(* CoDeSys 2.3.9.62 project: Cap11_7_Res.pro *)
(* Libraries: Standard.lib 4.10.05 12:14:46, IecSfc.lib*2.6.14 10:37:46 *)

(* Global variable list: Global_Variables *)
VAR_GLOBAL

 (* Entradas *)
	M: BOOL;

      (*Salidas*)
	Rojo: BOOL;    	(* Luz roja*)
	Amarillo:BOOL;	(* Luz amarilla *)
	Verde:BOOL;		(* Luz verde *)

END_VAR

(* POU PLC_PRG, SFC *)
PROGRAM PLC_PRG
VAR

       (* declaración  de temporizadores *)
	TEM_ROJO: TON;
	TEM_AMA: TON;
	TEM_VERDE: TON;

    (* declaración  de contadores *)
	CONTA: CTU;

       (* Variables auxiliares *)
	TVERDE: BOOL;     	(* Fin de temporizazión luz verde *)
	TAMA: BOOL;			(* Fin de temporizazión luz amarillo *)
	TROJO: BOOL;		(* Fin de temporizazión luz roja *)

	valor: INT:=3;			(* Número de ciclos a realizar antes de apagarse *)
END_VAR
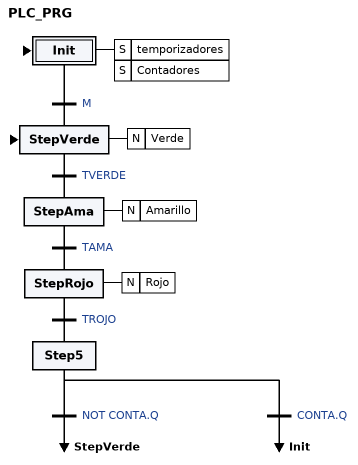
INITIAL_STEP Init:
	temporizadores(S);
	Contadores(S);
END_STEP
TRANSITION FROM Init TO StepVerde := M;
END_TRANSITION
STEP StepVerde:
	Verde(N);
END_STEP
TRANSITION FROM StepVerde TO StepAma := TVERDE;
END_TRANSITION
STEP StepAma:
	Amarillo(N);
END_STEP
TRANSITION FROM StepAma TO StepRojo := TAMA;
END_TRANSITION
STEP StepRojo:
	Rojo(N);
END_STEP
TRANSITION FROM StepRojo TO Step5 := TROJO;
END_TRANSITION
STEP Step5:
END_STEP
TRANSITION FROM Step5 TO StepVerde := NOT CONTA.Q;
END_TRANSITION
TRANSITION FROM Step5 TO Init := CONTA.Q;
END_TRANSITION
END_PROGRAM
ACTION Contadores:
	CAL		CONTA(CU:=StepVerde.x, RESET:=Init.x,PV:=valor)
END_ACTION
ACTION temporizadores:
	CAL		TEM_ROJO(IN:=StepRojo.x, PT:=T#5s, Q=>TROJO)

	CAL		TEM_AMA(IN:=StepAma.x, PT:=T#2s,Q=>TAMA)


	LD		StepVerde.x
	ST		TEM_VERDE.IN
	LD		T#2s
	ST		TEM_VERDE.PT
	CAL		TEM_VERDE
	LD		TEM_VERDE.Q
	ST		TVERDE
END_ACTION

(* Visualisation SemaforoSimple
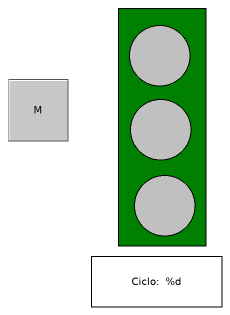
ellipse at (156,41)-(217,102): alarm colour if Rojo
ellipse at (157,115)-(218,176): alarm colour if Amarillo
ellipse at (161,191)-(222,252): alarm colour if Verde
rectangle at (118,272)-(249,323): text "Ciclo:  %d"; shows PLC_PRG.CONTA.CV
button at (35,95)-(95,157): text "M"; taps M
1 more shapes without text or variables
*)
